{attribute 'linkalways'} 
{attribute 'no_explicit_call' := 'This FB is a CLASS and must be accessed using methods or properties'}
{attribute 'enable_dynamic_creation'}
FUNCTION_BLOCK FINAL MAX_UINT EXTENDS Node
VAR
	in1 : _UINT(0);
	in2 : _UINT(0);
	out : _UINT(0);
END_VAR

METHOD PUBLIC Clone : I_Node
VAR
	pNode : POINTER TO MAX_UINT;
END_VAR
pNode := __NEW(MAX_UINT);
Clone := pNode^;
END_METHOD

METHOD FB_init : BOOL
VAR_INPUT
	bInitRetains : BOOL; // if TRUE, the retain variables are initialized (warm start / cold start)
	bInCopyCode : BOOL;  // if TRUE, the instance afterwards gets moved into the copy code (online change)
END_VAR
AddInput('in1',THIS^.in1);
AddInput('in2',THIS^.in2);
AddOutput('out', THIS^.out);
END_METHOD

METHOD PROTECTED OnExecute
VAR
END_VAR
out.Value := MAX(in1.Value, in2.Value);
END_METHOD

END_FUNCTION_BLOCK

(* stored: Version 1.1.0.1, ProductVersion 3.1.4024.15
   POU MAX_UINT: Id {817693e9-02d6-492a-9377-41be4d74e777}, SpecialFunc None
   Folder Constructor: Id {6b9e96d9-02e4-4b50-beb3-076f53ea39f6}
   Method Clone: Id {d6b084f4-9291-443a-87e5-576b79156997}
   Method FB_init: Id {bb5dfef2-7e18-4aff-aad6-3acd57922418}
   Method OnExecute: Id {c6d8073b-2f59-4526-9da7-deabfda0b7d7} *)
